FUNCTION_BLOCK SuspendedUnifiedProgramState EXTENDS SuspendedProgramState
VAR
	{attribute 'OPC.UA.DA' := '0'}
	_ClassName : STRING := __POUNAME();
END_VAR

{attribute 'monitoring' := 'call'}
PROPERTY ClassName : STRING
GET
ClassName := _ClassName;
END_GET
END_PROPERTY

END_FUNCTION_BLOCK

(* stored: Version 1.1.0.1
   POU SuspendedUnifiedProgramState: Id {85442c87-f833-4bd1-b74e-e172d59e8337}, SpecialFunc None
   Property ClassName: Id {af4d3fe5-9445-404a-9835-8b1666770d72}
   Get Get: Id {47f5fdff-0d91-4d3f-8226-172464fd7076} *)
